// TIA Portal V20 export
// export: Created 2025-12-01T14:57:12.6756315Z, ExportSetting None, DisplayName Totally Integrated Automation Portal, DisplayVersion V20 Update 3, DisplayName TIA Portal Openness, DisplayVersion V20 Update 3, DisplayName TIA Portal Version Control Interface, DisplayVersion V20 Update 3, DisplayName STEP 7 Professional, DisplayVersion V20 Update 3, DisplayName STEP 7 Safety, DisplayVersion V20 Update 2, DisplayName WinCC Basic/Comfort/Advanced, DisplayVersion V20 Update 3, DisplayName WinCC Professional, DisplayVersion V20 Update 3, DisplayName WinCC Unified, DisplayVersion V20 Update 3
FUNCTION "FC817_EventosEnv_Reset" : Void   // FC817, LAD
{ S7_Optimized_Access := 'FALSE' }
AUTHOR : TRACKING
NAME : 20141014
VERSION : 4.0
// stored: AutoNumber false, SetENOAutomatically false
   VAR_INPUT
      NumJDT : UInt;
   END_VAR
   VAR_TEMP
      P_Eventos : DWord;
      DBEventos : Word;
      NumDBEventos : UInt;
      MaxBytes : UInt;
      NumBytes : UInt;
      InicioBucleMesas : UInt;
      FinalBulceMesas : UInt;
      MesaDeJDT02 : Bool;
      JDT02_Activo : Bool;
      NumMesa : UInt;
      NumeroUT : UInt;
      Offset : UInt;
      Valor : UDInt;
      ValorReturn : Int;
      Cero : Byte;
   END_VAR
BEGIN

NETWORK
TITLE = Inicializar
/////////////////////////////////////////////////////////////////////////////////////
/// Inicio --> Se esta en el  JDT02

      SET;
      R     #JDT02_Activo;

      L     "JDT1_NDB_EventosEmi";
      T     #DBEventos;
      T     #NumDBEventos;
      L     "JDT1_MaxBytes";
      T     #MaxBytes;

      L     "JDT1_InicioBucleMesas";  // Tamaño Bucles
      T     #InicioBucleMesas;
      L     "JDT1_FinalBucleMesas";
      T     #FinalBulceMesas;


      L     #NumJDT;
      L     2;
      <>I;
      JC    NoJDT02;

      SET;
      S     #JDT02_Activo;

      L     "JDT2_NDB_EventosEmi";
      T     #DBEventos;
      T     #NumDBEventos;
      L     "JDT2_MaxBytes";
      T     #MaxBytes;

      L     "JDT2_InicioBucleMesas";  // Tamaño Bucles
      T     #InicioBucleMesas;
      L     "JDT2_FinalBucleMesas";
      T     #FinalBulceMesas;

NoJDT02:NOP   0;

/// Inicio --> Se esta en el JDT 02
/////////////////////////////////////////////////////////////////////////////////////



NETWORK
TITLE = Generar Eventos de las UT's
// - Recorrer todas las Mesas Buscando UT'que necesiten generar Eventos
//   Dos bucles anidados Mesas y UT's dentro de las Mesas ( No se hace)
// - Recorrer todas las UT's (Se hace
/////////////////////////////////////////////////////////////////////////////////////
// --- Recorrer todas las Mesas

      L     #InicioBucleMesas;
      T     #NumMesa;

Inicio_BucleDeMesas:NOP   0;
///////////////////////////////////////////////////////////////////////////////////////
/// Mirar si esta defincido como mesa de tracking

      SET;
      AN    "DB850_DefinicionMesas".Mesa[#NumMesa].ConfigMesa.MesaPaso;
      AN    "DB850_DefinicionMesas".Mesa[#NumMesa].ConfigMesa.MesaCruce;
      AN    "DB850_DefinicionMesas".Mesa[#NumMesa].ConfigMesa.MesaMultiplesDestinos;
      AN    "DB850_DefinicionMesas".Mesa[#NumMesa].ConfigMesa.MesaTL;  // añadido para evento rearme Nieves 11/04/24
      JC    Siguiente_BucleDeMesas;


///////////////////////////////////////////////////////////////////////////////////////
/// Mirar Si pertenece al JDT

      SET;
      X     "DB850_DefinicionMesas".Mesa[#NumMesa].ConfigMesa.MesaDeJDT02;
      XN    #JDT02_Activo;  // JDT01 o JDT02 ?
      =     #MesaDeJDT02;

      SET;
      AN    #MesaDeJDT02;
      JC    Siguiente_BucleDeMesas;


///////////////////////////////////////////////////////////////////////////////////////
// --- Comprobar Si hay que Enviar Eventos

// --- Informacion por Evento de CHEQ de Mesa >>> Ocupacion
      SET;
      A     "DB831_Mesas".Mesas[#NumMesa].EventosInformarJdT.OcupacionDeMesa;
      JC    EnviarEvento_OcupacionDeMesa;

// --- Informacion por Evento de CHEQ de Mesa >>> Mckey
      SET;
      A     "DB831_Mesas".Mesas[#NumMesa].EventosInformarJdT.MckeysEnMesa;

      JC    EnviarEvento_MckeysEnMesa;

// --- Informacion por Evento de CHEQ de Mesa >>> Todo - Ocupacion y Mckey
      SET;
      A     "DB831_Mesas".Mesas[#NumMesa].EventosInformarJdT.TodoDeMesa;
      JC    EnviarEvento_TodoDeMesa;


// --- Información por evento de pulsacion de rearme EVEN

      SET;
      A     "DB831_Mesas".Mesas[#NumMesa].Memorias.Evento_rearme;
      JC    EnviarEvento_rearme;


// --- No Hay que Enviar Eventos
///////////////////////////////////////////////////////////////////////////////////////
///////////////////////////////////////////////////////////////////////////////////////


///////////////////////////////////////////////////////////////////////////////////////
// --- Continuar recorriendo el resto de Mesas

Siguiente_BucleDeMesas:NOP   0;
      L     #NumMesa;
      L     #FinalBulceMesas;
      >=I;
      JC    FinalFuncion;  // Ya no hay más UT's ?

      L     #NumMesa;  // +1, Para la Siguiente UT
      L     1;
      +I;
      T     #NumMesa;

      JU    Inicio_BucleDeMesas;  // Ir a mirar la siguiente UT



NETWORK
TITLE = Evento de Evento de Ocupacion de Mesa
EnviarEvento_OcupacionDeMesa:NOP   0;

///////////////////////////////////////////////////////////////////////////////////////
// ---   Formateo del Evento de Estado del Dispositivo
// ---   * Mirar si hay sitio para generar el nuevo evento
// ---       * Inicializo NumBytes y Puntero al DB de Eventos Generados
// ---       * Calcula el tamaño de bytes que hay en el DB de Eventos Generados
// ---       * Comprobar si hay sitio para un evento más
// ---   *  Formatear el evento de Estado de Inicio de Bucle  INI!
///////////////////////////////////////////////////////////////////////////////////////


///////////////////////////////////////////////////////////////////////////////////////
// --- Mirar si hay sitio para generar un evento más
      L     0;
      T     #NumBytes;  // Inicializo el numero de Bytes
      T     #P_Eventos;  // Inicializo el puntero de Eventos Generados

Inicio_BusquedaFinalEventos_OcupacionDeMesa:NOP   0;
      OPN   DB [#DBEventos];  // Calcula el tamaño de bytes que hay en el DB
      L     DBB [#P_Eventos];
      L     0;
      ==I;
      JC    Fin_BusquedaFinalEventos_OcupacionDeMesa;  // Buscamos el final del DB = 0

      OPN   DB [#DBEventos];
      L     DBB [#P_Eventos];
      L     ' ';
      ==I;
      JC    Fin_BusquedaFinalEventos_OcupacionDeMesa;  // Buscamos el final del DB = ' '

      L     #P_Eventos;  // Incremento de P#1.0
      L     P#1.0;
      +D;
      T     #P_Eventos;

      JU    Inicio_BusquedaFinalEventos_OcupacionDeMesa;  // Continuar con el siguiente posicion

Fin_BusquedaFinalEventos_OcupacionDeMesa:NOP   0;
      L     #P_Eventos;  // Sacamos el NumBytes Escritos
      SRD   3;
      T     #NumBytes;

      L     #NumBytes;  // Miramos si hay sitio
      L     #MaxBytes;  // Max. que se pueden emitir, parametro
      >I;
      JC    FinalFuncion;  // No se pueden generar más eventos



///////////////////////////////////////////////////////////////////////////////////////
// --- Formatear el evento
      L     #P_Eventos;
      LAR2;  // Puntero al DB de Eventos Generados

      TAR2;  // Mirar si es el primer evento de la lista
      L     0;
      ==I;
      JC    NoEsInicio_ListaDeEventos_OcupacionDeMesa;  // Es el primero

      OPN   DB [#DBEventos];
      L     ',';  // Separador entre eventos ','
      T     DBB [AR2, P#0.0];
      +AR2  P#1.0;

NoEsInicio_ListaDeEventos_OcupacionDeMesa:NOP   0;

///////////////////////////////////////////////////////////////////////////////
// --- Cuerpo del Evento
      OPN   DB [#DBEventos];  // DB de Eventos Generados (A Emitir)
      L     '{';  // Inicio de Evento '{'
      T     DBB [AR2, P#0.0];
      +AR2  P#1.0;

      L     'CHE!';  // Evento - CHE!
      T     DBD [AR2, P#0.0];
      +AR2  P#4.0;


///////////////////////////////////////////////////////////////////////////////
      L     '[';
      T     DBB [AR2, P#0.0];
      L     'TIPO';
      T     DBD [AR2, P#1.0];
      L     ']';  // Evento - Atributo Mckey '[TIPO]'
      T     DBB [AR2, P#5.0];
      +AR2  P#6.0;

      L     'MESA';
      T     DBD [AR2, P#0.0];
      +AR2  P#4.0;


///////////////////////////////////////////////////////////////////////////////
      OPN   DB [#DBEventos];
      L     '[';  // Evento - Atributo Mesa  '[NUME]'
      T     DBB [AR2, P#0.0];
      L     'NUME';
      T     DBD [AR2, P#1.0];
      L     ']';
      T     DBB [AR2, P#5.0];
      +AR2  P#6.0;

      L     #NumMesa;
      L     "CTE_OffsetMesa";
      +I;
      T     #Valor;

// --- Convertir Valor a ASCII -  Mesa Actual
      TAR2;
      SRD   3;
      T     #NumBytes;  // Miro que offset tiene la String

      CALL  "FC893_Obtener_StringDelAtributo"
      ( DB_String := #NumDBEventos,
        OffsetIni := #NumBytes,
        Valor     := #Valor,
        OffsetFin := #Offset
      );  // Llamo a ObtenerStrinAtributo

      L     #Offset;
      SLD   3;
      LAR2;  // Recupero que offset tiene la String
// --- Ya esta convertido el Valor a ASCI - Fin Mesa Actual



///////////////////////////////////////////////////////////////////////////////
      L     '[';
      T     DBB [AR2, P#0.0];
      L     'OPER';
      T     DBD [AR2, P#1.0];
      L     ']';  // Evento - Atributo Mckey '[TIPO]'
      T     DBB [AR2, P#5.0];
      +AR2  P#6.0;

      L     'OCUP';
      T     DBD [AR2, P#0.0];
      +AR2  P#4.0;


///////////////////////////////////////////////////////////////////////////////
      OPN   DB [#DBEventos];
      L     '[';  // Evento - Atributo Ocupacion '[OCUP]'
      T     DBB [AR2, P#0.0];
      L     'OCUP';
      T     DBD [AR2, P#1.0];
      L     ']';
      T     DBB [AR2, P#5.0];
      +AR2  P#6.0;

      L     'NO';  // No Ocupado

      SET;
      AN    "DB900_Estado_Mesas".EstadoVI[#NumMesa].En_PHS_1;
      AN    "DB900_Estado_Mesas".EstadoVI[#NumMesa].En_PHS_2;
      JC    NoOcupado_OcupacionDeMesa;

      L     'SI';  // Esta Ocupado

NoOcupado_OcupacionDeMesa:NOP   0;
      OPN   DB [#DBEventos];
      T     DBW [AR2, P#0.0];
      +AR2  P#2.0;


///////////////////////////////////////////////////////////////////////////////
      OPN   DB [#DBEventos];
      L     '[';  // Evento - Atributo Resultado'[RESU]'
      T     DBB [AR2, P#0.0];
      L     'RESU';
      T     DBD [AR2, P#1.0];
      L     ']';
      T     DBB [AR2, P#5.0];
      +AR2  P#6.0;

      L     'OK';
      T     DBW [AR2, P#0.0];
      +AR2  P#2.0;


///////////////////////////////////////////////////////////////////////////////
// --- Final del Evento

      OPN   DB [#DBEventos];  // DB de Eventos Generados (A Emitir)
      L     '}';  // --- Fin de Evento '}'
      T     DBB [AR2, P#0.0];
      +AR2  P#1.0;


///////////////////////////////////////////////////////////////////////////////
/// -- Dar  por enviado el evento

      SET;
      R     "DB831_Mesas".Mesas[#NumMesa].EventosInformarJdT.OcupacionDeMesa;

      JU    Siguiente_BucleDeMesas;



NETWORK
TITLE = Evento de Evento de Mckeys En Mesa
EnviarEvento_MckeysEnMesa:NOP   0;

///////////////////////////////////////////////////////////////////////////////////////
// ---   Formateo del Evento de Estado del Dispositivo
// ---   * Mirar si hay sitio para generar el nuevo evento
// ---       * Inicializo NumBytes y Puntero al DB de Eventos Generados
// ---       * Calcula el tamaño de bytes que hay en el DB de Eventos Generados
// ---       * Comprobar si hay sitio para un evento más
// ---   *  Formatear el evento de Estado de Inicio de Bucle  INI!
///////////////////////////////////////////////////////////////////////////////////////


///////////////////////////////////////////////////////////////////////////////////////
// --- Mirar si hay sitio para generar un evento más
      L     0;
      T     #NumBytes;  // Inicializo el numero de Bytes
      T     #P_Eventos;  // Inicializo el puntero de Eventos Generados

Inicio_BusquedaFinalEventos_MckeysEnMesa:NOP   0;
      OPN   DB [#DBEventos];  // Calcula el tamaño de bytes que hay en el DB
      L     DBB [#P_Eventos];
      L     0;
      ==I;
      JC    Fin_BusquedaFinalEventos_MckeysEnMesa;  // Buscamos el final del DB = 0

      OPN   DB [#DBEventos];
      L     DBB [#P_Eventos];
      L     ' ';
      ==I;
      JC    Fin_BusquedaFinalEventos_MckeysEnMesa;  // Buscamos el final del DB = ' '

      L     #P_Eventos;  // Incremento de P#1.0
      L     P#1.0;
      +D;
      T     #P_Eventos;

      JU    Inicio_BusquedaFinalEventos_MckeysEnMesa;  // Continuar con el siguiente posicion

Fin_BusquedaFinalEventos_MckeysEnMesa:NOP   0;
      L     #P_Eventos;  // Sacamos el NumBytes Escritos
      SRD   3;
      T     #NumBytes;

      L     #NumBytes;  // Miramos si hay sitio
      L     #MaxBytes;  // Max. que se pueden emitir, parametro
      >I;
      JC    FinalFuncion;  // No se pueden generar más eventos



///////////////////////////////////////////////////////////////////////////////////////
// --- Formatear el evento
      L     #P_Eventos;
      LAR2;  // Puntero al DB de Eventos Generados

      TAR2;  // Mirar si es el primer evento de la lista
      L     0;
      ==I;
      JC    NoEsInicio_ListaDeEventos_MckeysEnMesa;  // Es el primero

      OPN   DB [#DBEventos];
      L     ',';  // Separador entre eventos ','
      T     DBB [AR2, P#0.0];
      +AR2  P#1.0;

NoEsInicio_ListaDeEventos_MckeysEnMesa:NOP   0;

///////////////////////////////////////////////////////////////////////////////
// --- Cuerpo del Evento
      OPN   DB [#DBEventos];  // DB de Eventos Generados (A Emitir)
      L     '{';  // Inicio de Evento '{'
      T     DBB [AR2, P#0.0];
      +AR2  P#1.0;

      L     'CHE!';  // Evento - CHE!
      T     DBD [AR2, P#0.0];
      +AR2  P#4.0;


///////////////////////////////////////////////////////////////////////////////
      L     '[';
      T     DBB [AR2, P#0.0];
      L     'TIPO';
      T     DBD [AR2, P#1.0];
      L     ']';  // Evento - Atributo Mckey '[TIPO]'
      T     DBB [AR2, P#5.0];
      +AR2  P#6.0;

      L     'MESA';
      T     DBD [AR2, P#0.0];
      +AR2  P#4.0;


///////////////////////////////////////////////////////////////////////////////
      OPN   DB [#DBEventos];
      L     '[';  // Evento - Atributo Mesa  '[NUME]'
      T     DBB [AR2, P#0.0];
      L     'NUME';
      T     DBD [AR2, P#1.0];
      L     ']';
      T     DBB [AR2, P#5.0];
      +AR2  P#6.0;

      L     #NumMesa;
      L     "CTE_OffsetMesa";
      +I;
      T     #Valor;

// --- Convertir Valor a ASCII -  Mesa Actual
      TAR2;
      SRD   3;
      T     #NumBytes;  // Miro que offset tiene la String

      CALL  "FC893_Obtener_StringDelAtributo"
      ( DB_String := #NumDBEventos,
        OffsetIni := #NumBytes,
        Valor     := #Valor,
        OffsetFin := #Offset
      );  // Llamo a ObtenerStrinAtributo

      L     #Offset;
      SLD   3;
      LAR2;  // Recupero que offset tiene la String
// --- Ya esta convertido el Valor a ASCI - Fin Mesa Actual



///////////////////////////////////////////////////////////////////////////////
      L     '[';
      T     DBB [AR2, P#0.0];
      L     'OPER';
      T     DBD [AR2, P#1.0];
      L     ']';  // Evento - Atributo Mckey '[TIPO]'
      T     DBB [AR2, P#5.0];
      +AR2  P#6.0;

      L     'MCKY';
      T     DBD [AR2, P#0.0];
      +AR2  P#4.0;


///////////////////////////////////////////////////////////////////////////////
      OPN   DB [#DBEventos];
      L     '[';  // Evento - Atributo Mckeys '[MCKY]'
      T     DBB [AR2, P#0.0];
      L     'MCKY';
      T     DBD [AR2, P#1.0];
      L     ']';
      T     DBB [AR2, P#5.0];
      +AR2  P#6.0;

// ---- Inicio de Mckeys
      OPN   DB [#DBEventos];
      L     '(';
      T     DBB [AR2, P#0.0];
      +AR2  P#1.0;

// --- Bucle de Mckeys >>> Hay Una UT
      L     "DB810_ColasMesas".Colas[#NumMesa].UT_PrimeraMesa;
      T     #NumeroUT;

      SET;  // Hay UT ?
      L     #NumeroUT;
      L     0;
      ==I;
      JC    FinalBucleUTs_MckeysEnMesa;

      L     "DB812_UTs_Control".UT[#NumeroUT].Mckey;
      T     #Valor;

// --- Convertir Valor a ASCII -  Mesa Actual
      TAR2;
      SRD   3;
      T     #NumBytes;  // Miro que offset tiene la String

      CALL  "FC893_Obtener_StringDelAtributo"
      ( DB_String := #NumDBEventos,
        OffsetIni := #NumBytes,
        Valor     := #Valor,
        OffsetFin := #Offset
      );  // Llamo a ObtenerStrinAtributo

      L     #Offset;
      SLD   3;
      LAR2;  // Recupero que offset tiene la String
// --- Ya esta convertido el Valor a ASCI - Fin Mesa Actual

      L     "DB812_UTs_Control".UT[#NumeroUT].UT_SiguienteMesa;
      T     #NumeroUT;

// --- Bucle de Mckeys >>> Hay Mas UTs
IncioBucleUTs_MckeysEnMesa:NOP   0;
      SET;  // Hay UT ?
      L     #NumeroUT;
      L     0;
      ==I;
      JC    FinalBucleUTs_MckeysEnMesa;

      OPN   DB [#DBEventos];
      L     ',';  // Separador de Mckeys
      T     DBB [AR2, P#0.0];
      +AR2  P#1.0;

      L     "DB812_UTs_Control".UT[#NumeroUT].Mckey;
      T     #Valor;

// --- Convertir Valor a ASCII -  Mesa Actual
      TAR2;
      SRD   3;
      T     #NumBytes;  // Miro que offset tiene la String

      CALL  "FC893_Obtener_StringDelAtributo"
      ( DB_String := #NumDBEventos,
        OffsetIni := #NumBytes,
        Valor     := #Valor,
        OffsetFin := #Offset
      );  // Llamo a ObtenerStrinAtributo

      L     #Offset;
      SLD   3;
      LAR2;  // Recupero que offset tiene la String
// --- Ya esta convertido el Valor a ASCI - Fin Mesa Actual


      L     "DB812_UTs_Control".UT[#NumeroUT].UT_SiguienteMesa;
      T     #NumeroUT;
      JU    IncioBucleUTs_MckeysEnMesa;

FinalBucleUTs_MckeysEnMesa:NOP   0;

// --- Final de Mckeys
      OPN   DB [#DBEventos];
      L     ')';
      T     DBB [AR2, P#0.0];
      +AR2  P#1.0;


///////////////////////////////////////////////////////////////////////////////
      OPN   DB [#DBEventos];
      L     '[';  // Evento - Atributo Resultado'[RESU]'
      T     DBB [AR2, P#0.0];
      L     'RESU';
      T     DBD [AR2, P#1.0];
      L     ']';
      T     DBB [AR2, P#5.0];
      +AR2  P#6.0;

      L     'OK';
      T     DBW [AR2, P#0.0];
      +AR2  P#2.0;


///////////////////////////////////////////////////////////////////////////////
// --- Final del Evento

      OPN   DB [#DBEventos];  // DB de Eventos Generados (A Emitir)
      L     '}';  // --- Fin de Evento '}'
      T     DBB [AR2, P#0.0];
      +AR2  P#1.0;


///////////////////////////////////////////////////////////////////////////////
/// -- Dar  por enviado el evento

      SET;
      R     "DB831_Mesas".Mesas[#NumMesa].EventosInformarJdT.MckeysEnMesa;

      JU    Siguiente_BucleDeMesas;



NETWORK
TITLE = Evento de Evento de Todo De Mesa >>> Ocupacion, Mckeys
EnviarEvento_TodoDeMesa:NOP   0;

///////////////////////////////////////////////////////////////////////////////////////
// ---   Formateo del Evento de Estado del Dispositivo
// ---   * Mirar si hay sitio para generar el nuevo evento
// ---       * Inicializo NumBytes y Puntero al DB de Eventos Generados
// ---       * Calcula el tamaño de bytes que hay en el DB de Eventos Generados
// ---       * Comprobar si hay sitio para un evento más
// ---   *  Formatear el evento de Estado de Inicio de Bucle  INI!
///////////////////////////////////////////////////////////////////////////////////////


///////////////////////////////////////////////////////////////////////////////////////
// --- Mirar si hay sitio para generar un evento más
      L     0;
      T     #NumBytes;  // Inicializo el numero de Bytes
      T     #P_Eventos;  // Inicializo el puntero de Eventos Generados

Inicio_BusquedaFinalEventos_TodoDeMesa:NOP   0;
      OPN   DB [#DBEventos];  // Calcula el tamaño de bytes que hay en el DB
      L     DBB [#P_Eventos];
      L     0;
      ==I;
      JC    Fin_BusquedaFinalEventos_TodoDeMesa;  // Buscamos el final del DB = 0

      OPN   DB [#DBEventos];
      L     DBB [#P_Eventos];
      L     ' ';
      ==I;
      JC    Fin_BusquedaFinalEventos_TodoDeMesa;  // Buscamos el final del DB = ' '

      L     #P_Eventos;  // Incremento de P#1.0
      L     P#1.0;
      +D;
      T     #P_Eventos;

      JU    Inicio_BusquedaFinalEventos_TodoDeMesa;  // Continuar con el siguiente posicion

Fin_BusquedaFinalEventos_TodoDeMesa:NOP   0;
      L     #P_Eventos;  // Sacamos el NumBytes Escritos
      SRD   3;
      T     #NumBytes;

      L     #NumBytes;  // Miramos si hay sitio
      L     #MaxBytes;  // Max. que se pueden emitir, parametro
      >I;
      JC    FinalFuncion;  // No se pueden generar más eventos



///////////////////////////////////////////////////////////////////////////////////////
// --- Formatear el evento
      L     #P_Eventos;
      LAR2;  // Puntero al DB de Eventos Generados

      TAR2;  // Mirar si es el primer evento de la lista
      L     0;
      ==I;
      JC    NoEsInicio_ListaDeEventos_TodoDeMesa;  // Es el primero

      OPN   DB [#DBEventos];
      L     ',';  // Separador entre eventos ','
      T     DBB [AR2, P#0.0];
      +AR2  P#1.0;

NoEsInicio_ListaDeEventos_TodoDeMesa:NOP   0;

///////////////////////////////////////////////////////////////////////////////
// --- Cuerpo del Evento
      OPN   DB [#DBEventos];  // DB de Eventos Generados (A Emitir)
      L     '{';  // Inicio de Evento '{'
      T     DBB [AR2, P#0.0];
      +AR2  P#1.0;

      L     'CHE!';  // Evento - CHE!
      T     DBD [AR2, P#0.0];
      +AR2  P#4.0;


///////////////////////////////////////////////////////////////////////////////
      L     '[';
      T     DBB [AR2, P#0.0];
      L     'TIPO';
      T     DBD [AR2, P#1.0];
      L     ']';  // Evento - Atributo Mckey '[TIPO]'
      T     DBB [AR2, P#5.0];
      +AR2  P#6.0;

      L     'MESA';
      T     DBD [AR2, P#0.0];
      +AR2  P#4.0;


///////////////////////////////////////////////////////////////////////////////
      OPN   DB [#DBEventos];
      L     '[';  // Evento - Atributo Mesa  '[NUME]'
      T     DBB [AR2, P#0.0];
      L     'NUME';
      T     DBD [AR2, P#1.0];
      L     ']';
      T     DBB [AR2, P#5.0];
      +AR2  P#6.0;

      L     #NumMesa;
      L     "CTE_OffsetMesa";
      +I;
      T     #Valor;

// --- Convertir Valor a ASCII -  Mesa Actual
      TAR2;
      SRD   3;
      T     #NumBytes;  // Miro que offset tiene la String

      CALL  "FC893_Obtener_StringDelAtributo"
      ( DB_String := #NumDBEventos,
        OffsetIni := #NumBytes,
        Valor     := #Valor,
        OffsetFin := #Offset
      );  // Llamo a ObtenerStrinAtributo

      L     #Offset;
      SLD   3;
      LAR2;  // Recupero que offset tiene la String
// --- Ya esta convertido el Valor a ASCI - Fin Mesa Actual



///////////////////////////////////////////////////////////////////////////////
      L     '[';
      T     DBB [AR2, P#0.0];
      L     'OPER';
      T     DBD [AR2, P#1.0];
      L     ']';  // Evento - Atributo Mckey '[TIPO]'
      T     DBB [AR2, P#5.0];
      +AR2  P#6.0;

      L     'TODO';
      T     DBD [AR2, P#0.0];
      +AR2  P#4.0;


///////////////////////////////////////////////////////////////////////////////
      OPN   DB [#DBEventos];
      L     '[';  // Evento - Atributo Mckeys '[MCKY]'
      T     DBB [AR2, P#0.0];
      L     'MCKY';
      T     DBD [AR2, P#1.0];
      L     ']';
      T     DBB [AR2, P#5.0];
      +AR2  P#6.0;

// ---- Inicio de Mckeys
      OPN   DB [#DBEventos];
      L     '(';
      T     DBB [AR2, P#0.0];
      +AR2  P#1.0;

// --- Bucle de Mckeys >>> Hay Una UT
      L     "DB810_ColasMesas".Colas[#NumMesa].UT_PrimeraMesa;
      T     #NumeroUT;

      SET;  // Hay UT ?
      L     #NumeroUT;
      L     0;
      ==I;
      JC    FinalBucleUTs_TodoDeMesa;

      L     "DB812_UTs_Control".UT[#NumeroUT].Mckey;
      T     #Valor;

// --- Convertir Valor a ASCII -  Mesa Actual
      TAR2;
      SRD   3;
      T     #NumBytes;  // Miro que offset tiene la String

      CALL  "FC893_Obtener_StringDelAtributo"
      ( DB_String := #NumDBEventos,
        OffsetIni := #NumBytes,
        Valor     := #Valor,
        OffsetFin := #Offset
      );  // Llamo a ObtenerStrinAtributo

      L     #Offset;
      SLD   3;
      LAR2;  // Recupero que offset tiene la String
// --- Ya esta convertido el Valor a ASCI - Fin Mesa Actual

      L     "DB812_UTs_Control".UT[#NumeroUT].UT_SiguienteMesa;
      T     #NumeroUT;

// --- Bucle de Mckeys >>> Hay Mas UTs
IncioBucleUTs_TodoDeMesa:NOP   0;
      SET;  // Hay UT ?
      L     #NumeroUT;
      L     0;
      ==I;
      JC    FinalBucleUTs_TodoDeMesa;

      OPN   DB [#DBEventos];
      L     ',';  // Separador de Mckeys
      T     DBB [AR2, P#0.0];
      +AR2  P#1.0;

      L     "DB812_UTs_Control".UT[#NumeroUT].Mckey;
      T     #Valor;

// --- Convertir Valor a ASCII -  Mesa Actual
      TAR2;
      SRD   3;
      T     #NumBytes;  // Miro que offset tiene la String

      CALL  "FC893_Obtener_StringDelAtributo"
      ( DB_String := #NumDBEventos,
        OffsetIni := #NumBytes,
        Valor     := #Valor,
        OffsetFin := #Offset
      );  // Llamo a ObtenerStrinAtributo

      L     #Offset;
      SLD   3;
      LAR2;  // Recupero que offset tiene la String
// --- Ya esta convertido el Valor a ASCI - Fin Mesa Actual


      L     "DB812_UTs_Control".UT[#NumeroUT].UT_SiguienteMesa;
      T     #NumeroUT;
      JU    IncioBucleUTs_TodoDeMesa;

FinalBucleUTs_TodoDeMesa:NOP   0;





// --- Final de Mckeys
      OPN   DB [#DBEventos];
      L     ')';
      T     DBB [AR2, P#0.0];
      +AR2  P#1.0;


///////////////////////////////////////////////////////////////////////////////
      OPN   DB [#DBEventos];
      L     '[';  // Evento - Atributo Ocupacion '[OCUP]'
      T     DBB [AR2, P#0.0];
      L     'OCUP';
      T     DBD [AR2, P#1.0];
      L     ']';
      T     DBB [AR2, P#5.0];
      +AR2  P#6.0;

      L     'NO';  // No Ocupado

      SET;
      AN    "DB900_Estado_Mesas".EstadoVI[#NumMesa].En_PHS_1;
      AN    "DB900_Estado_Mesas".EstadoVI[#NumMesa].En_PHS_2;
      JC    NoOcupado_TodoDeMesa;

      L     'SI';  // Esta Ocupado

NoOcupado_TodoDeMesa:NOP   0;
      OPN   DB [#DBEventos];
      T     DBW [AR2, P#0.0];
      +AR2  P#2.0;


///////////////////////////////////////////////////////////////////////////////
      OPN   DB [#DBEventos];
      L     '[';  // Evento - Atributo Resultado'[RESU]'
      T     DBB [AR2, P#0.0];
      L     'RESU';
      T     DBD [AR2, P#1.0];
      L     ']';
      T     DBB [AR2, P#5.0];
      +AR2  P#6.0;

      L     'OK';
      T     DBW [AR2, P#0.0];
      +AR2  P#2.0;


///////////////////////////////////////////////////////////////////////////////
// --- Final del Evento

      OPN   DB [#DBEventos];  // DB de Eventos Generados (A Emitir)
      L     '}';  // --- Fin de Evento '}'
      T     DBB [AR2, P#0.0];
      +AR2  P#1.0;


///////////////////////////////////////////////////////////////////////////////
/// -- Dar  por enviado el evento

      SET;
      R     "DB831_Mesas".Mesas[#NumMesa].EventosInformarJdT.TodoDeMesa;

      JU    Siguiente_BucleDeMesas;



NETWORK
TITLE = Emision de Evento Rearme
EnviarEvento_rearme:NOP   0;

///////////////////////////////////////////////////////////////////////////////////////
// ---   Formateo del Evento de Estado del Dispositivo
// ---   * Mirar si hay sitio para generar el nuevo evento
// ---       * Inicializo NumBytes y Puntero al DB de Eventos Generados
// ---       * Calcula el tamaño de bytes que hay en el DB de Eventos Generados
// ---       * Comprobar si hay sitio para un evento más
// ---   *  Formatear el evento de Estado de Inicio de Bucle
///////////////////////////////////////////////////////////////////////////////////////

// --- Primero miramos si tenemos configurado emitir el evento o no
      SET;
      A     "DB831_Mesas".Mesas[#NumMesa].EventosInformarJdT.Evento_Rearme;
      JC    emite_evento_rearme;

      SET;
      R     "DB831_Mesas".Mesas[#NumMesa].Memorias.Evento_rearme;
      JC    Siguiente_BucleDeMesas;

///////////////////////////////////////////////////////////////////////////////////////
// --- Mirar si hay sitio para generar un evento más
emite_evento_rearme:NOP   0;
      L     0;
      T     #NumBytes;  // Inicializo el numero de Bytes
      T     #P_Eventos;  // Inicializo el puntero de Eventos Generados

Inicio_BusquedaFinalEventos_rearme:NOP   0;
      OPN   DB [#DBEventos];  // Calcula el tamaño de bytes que hay en el DB
      L     DBB [#P_Eventos];
      L     0;
      ==I;
      JC    Fin_BusquedaFinalEventos_rearme;  // Buscamos el final del DB = 0

      OPN   DB [#DBEventos];
      L     DBB [#P_Eventos];
      L     ' ';
      ==I;
      JC    Fin_BusquedaFinalEventos_rearme;  // Buscamos el final del DB = ' '

      L     #P_Eventos;  // Incremento de P#1.0
      L     P#1.0;
      +D;
      T     #P_Eventos;

      JU    Inicio_BusquedaFinalEventos_rearme;  //Continuar con el siguiente posicion

Fin_BusquedaFinalEventos_rearme:NOP   0;
      L     #P_Eventos;  // Sacamos el NumBytes Escritos
      SRD   3;
      T     #NumBytes;

      L     #NumBytes;  // Miramos si hay sitio
      L     #MaxBytes;  // Max. que se pueden emitir, parametro
      >I;
      JC    FinalFuncion;  // No se pueden generar más eventos



///////////////////////////////////////////////////////////////////////////////////////
// --- Formatear el evento
      L     #P_Eventos;
      LAR2;  // Puntero al DB de Eventos Generados

      TAR2;  // Mirar si es el primer evento de la lista
      L     0;
      ==I;
      JC    NoEsInicio_ListaDeEventos_rearme;  // Es el primero

      OPN   DB [#DBEventos];
      L     ',';  // Separador entre eventos ','
      T     DBB [AR2, P#0.0];
      +AR2  P#1.0;

NoEsInicio_ListaDeEventos_rearme:NOP   0;

///////////////////////////////////////////////////////////////////////////////
// --- Cuerpo del Evento
      OPN   DB [#DBEventos];  // DB de Eventos Generados (A Emitir)
      L     '{';  // Inicio de Evento '{'
      T     DBB [AR2, P#0.0];
      +AR2  P#1.0;

      L     'EVEN';  // Evento - EVEN
      T     DBD [AR2, P#0.0];
      +AR2  P#4.0;


///////////////////////////////////////////////////////////////////////////////
      L     '[';
      T     DBB [AR2, P#0.0];
      L     'TIPO';
      T     DBD [AR2, P#1.0];
      L     ']';  // Evento - Atributo Mckey '[TIPO]'
      T     DBB [AR2, P#5.0];
      +AR2  P#6.0;

      L     'MESA';
      T     DBD [AR2, P#0.0];
      +AR2  P#4.0;


///////////////////////////////////////////////////////////////////////////////
      OPN   DB [#DBEventos];
      L     '[';  // Evento - Atributo Mesa  '[NUME]'
      T     DBB [AR2, P#0.0];
      L     'NUME';
      T     DBD [AR2, P#1.0];
      L     ']';
      T     DBB [AR2, P#5.0];
      +AR2  P#6.0;

      L     #NumMesa;
      L     "CTE_OffsetMesa";
      +I;
      T     #Valor;

// --- Convertir Valor a ASCII -  Mesa Actual
      TAR2;
      SRD   3;
      T     #NumBytes;  // Miro que offset tiene la String

      CALL  "FC893_Obtener_StringDelAtributo"
      ( DB_String := #NumDBEventos,
        OffsetIni := #NumBytes,
        Valor     := #Valor,
        OffsetFin := #Offset
      );  // Llamo a ObtenerStrinAtributo

      L     #Offset;
      SLD   3;
      LAR2;  // Recupero que offset tiene la String
// --- Ya esta convertido el Valor a ASCI - Fin Mesa Actual



///////////////////////////////////////////////////////////////////////////////
      L     '[';
      T     DBB [AR2, P#0.0];
      L     'OPER';
      T     DBD [AR2, P#1.0];
      L     ']';  // Evento - Atributo Mckey '[TIPO]'
      T     DBB [AR2, P#5.0];
      +AR2  P#6.0;

      L     'REAR';
      T     DBD [AR2, P#0.0];
      +AR2  P#4.0;


///////////////////////////////////////////////////////////////////////////////
// --- Final del Evento

      OPN   DB [#DBEventos];  // DB de Eventos Generados (A Emitir)
      L     '}';  // --- Fin de Evento '}'
      T     DBB [AR2, P#0.0];
      +AR2  P#1.0;


///////////////////////////////////////////////////////////////////////////////
/// -- Dar  por enviado el evento

      SET;
      R     "DB831_Mesas".Mesas[#NumMesa].Memorias.Evento_rearme;

      JU    Siguiente_BucleDeMesas;



NETWORK
TITLE = Final de la Función
/////////////////////////////////////////////////////////////////////////////////////
FinalFuncion:NOP   0;


END_FUNCTION
